PROGRAM P_Output
VAR
	fbOneValveOutput 	: FB_OutputNormalizing;
	fbTwoValveOutput 	: FB_OutputNormalizing;
END_VAR

fbOneValveOutput(
	fNormalizedInput := G_OPC.fValveOneOutput,
	bEnable := (G_Enables.bEnableU AND G_Enables.bEnableOne),
	nOutput => G_Output.nValveOneOutput	
);

fbTwoValveOutput(
	fNormalizedInput := G_OPC.fValveTwoOutput,
	bEnable := (G_Enables.bEnableU AND G_Enables.bEnableTwo),
	nOutput => G_Output.nValveTwoOutput	
);

END_PROGRAM

(* stored: Version 1.1.0.1
   POU P_Output: Id {ea868c64-71e1-491f-a495-e9db7d8a4d4c}, SpecialFunc None *)
